PROGRAM P_Demo_FB_DMXGetLampOnMode
VAR
    fbGetLampOnMode   : FB_DMXGetLampOnMode;          // 读开灯模式
    stDmxCmdBuffer    : ST_DMXCommandBuffer;          // 与通讯 FB 共用
    wTargetManufId    : WORD := 16#4241;              // 目标灯具厂商 ID
    dwTargetDeviceId  : DWORD := 16#12131415;         // 目标灯具设备 ID
    byTargetPort      : BYTE := 0;                    // 根设备通道 0
    bDoRead           : BOOL := FALSE;                // 在线给一次上升沿触发
    bBusy             : BOOL;
    bError            : BOOL;
    udiErrId          : UDINT;
    eOnMode           : E_DMXLampOnMode;              // 当前开灯模式
END_VAR

// ============================================================
// Tc2_DMX.FB_DMXGetLampOnMode 演示程序
// ============================================================
// 场景：调试灯具上电行为：核对每盏灯当前开灯模式是否符合现场要求（如收到 DMX 数据后才亮）。
// 价值：把开灯行为参数读进 PLC，便于在 HMI 集中核对/显示，无需逐台进设备菜单查看。
// 验证：给 bDoRead 一次上升沿 -> bBusy 短暂 TRUE -> 回 FALSE 后 eOnMode 即设备当前开灯模式枚举值。
// 验证步骤：
//   1. 右键 PLC 项目下 POUs 文件夹 → Add → Existing Item → 选本 .TcPOU 文件
//   2. 引用 Tc2_DMX；同项目里放一个 FB_EL6851CommunicationEx 实例并共用 stDmxCmdBuffer（非 CycleMode）
//   3. 编译 → 登录 → 运行；按上方『验证』行在线给上升沿观察
// ============================================================

fbGetLampOnMode(
    bStart                     := bDoRead,
    wDestinationManufacturerId := wTargetManufId,
    dwDestinationDeviceId      := dwTargetDeviceId,
    byPortId                   := byTargetPort,
    dwOptions                  := 0,
    stCommandBuffer            := stDmxCmdBuffer,
    bBusy                      => bBusy,
    bError                     => bError,
    udiErrorId                 => udiErrId,
    eLampOnMode                => eOnMode
);

END_PROGRAM

(* stored: Version 1.1.0.1, ProductVersion 3.1.4024.5
   POU P_Demo_FB_DMXGetLampOnMode: Id {04748319-712b-5479-b168-8839ce04d53b}, SpecialFunc None *)
